// Mitsubishi GX Works2 project: 실린더응용1   PLC: Q02/Q02H

PROGRAM MAIN
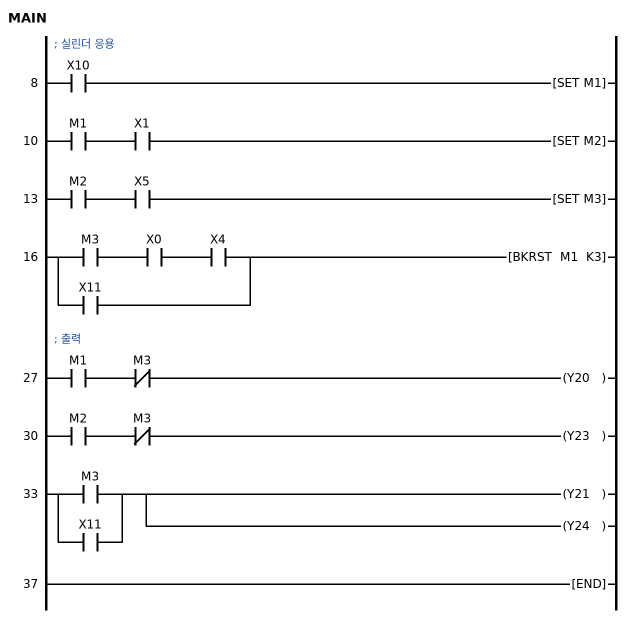
; 실린더 응용
8     LD      X10
      SET     M1
10    LD      M1
      AND     X1
      SET     M2
13    LD      M2
      AND     X5
      SET     M3
16    LD      M3
      AND     X0
      AND     X4
      OR      X11
      BKRST   M1 K3
; 출력
27    LD      M1
      ANI     M3
      OUT     Y20
30    LD      M2
      ANI     M3
      OUT     Y23
33    LD      M3
      OR      X11
      OUT     Y21
      OUT     Y24
37    END
END_PROGRAM
